Fanuc KAREL source: compact_preamble.KL

PROGRAM KB00177
%NOLOCKGROUP
VAR
P1:INTEGER;P2:INTEGER;P3 : XYZWPR;P4:INTEGER
BEGIN
P1=1
P2=1
P3.X=1.0
P4=1
SET_POS_TPE(P1,P2,P3,P4,1)
END KB00177
